TYPE "UDT_ZC_CONTADOR_TIEMPO"
TITLE = ZC_CONTADOR_TIEMPO_V1_0
VERSION : 0.1
//Tipo de dato contador tiempo
   STRUCT
      Hora : UDInt;   // Contador Horas
      Minuto : USInt;   // Contador Minutos
      Segundo : USInt;   // Contador Segundos
   END_STRUCT;

END_TYPE

